TYPE TurnTableOutput :
STRUCT
	
o_TurnTable_REF_SENSOR:BOOL;
o_TurnTable_FWD_SENSOR:BOOL;
o_TurnTable_REV_SENSOR:BOOL;
END_STRUCT

END_TYPE

(* stored: Version 1.1.0.1, ProductVersion 3.1.4024.16
   DUT TurnTableOutput: Id {7dc23f69-d91b-49d4-ad02-bd49b23c2110} *)
